(* CoDeSys 2.3 export: ATTIC.EXP *)

(* POU Rooms/Attic, ST *)
FUNCTION_BLOCK Attic
VAR
END_VAR
;
END_FUNCTION_BLOCK
